KUKA KRL program: SAMPLE.SRC

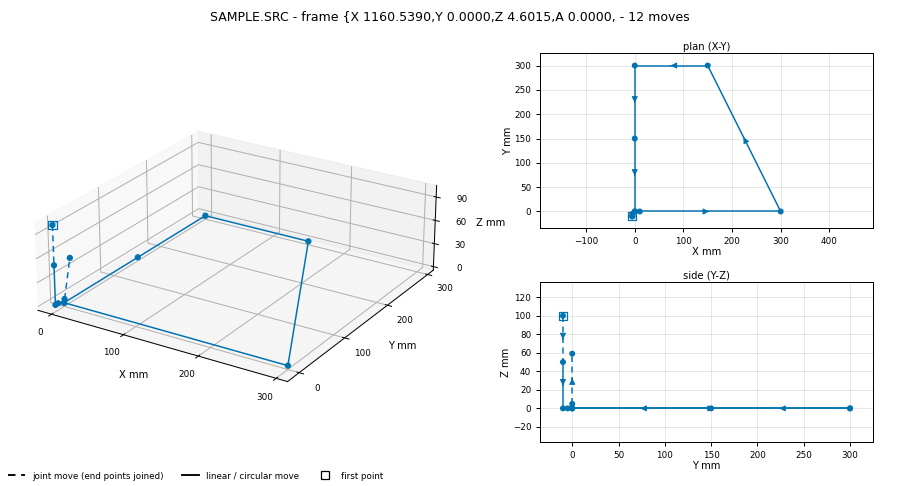
[picture p0: tool path of SAMPLE.SRC in frame {X 1160.5390,Y 0.0000,Z 4.6015,A 0.0000,, 12 of 14 moves have a stored position in this frame; points joined in program order, loops and branches not executed]
&ACCESS RVP
&REL 1
&COMMENT GENERATED BY ROBOTMASTER
&PARAM TEMPLATE = C:\KRC\Roboter\Template\vorgabe
&PARAM EDITMASK = *
DEF BTEST()

EXT BAS (BAS_COMMAND :IN,REAL :IN )
EXT TOOL(INT:IN)
EXT TOOLON()
EXT TOOLOFF()

INT I
BAS (#INITMOV,0 )

;******SETTINGS FOR PTP MOTION***********************
;FOLD
;SET PTP $VEL_AXIS AND $ACC_AXIS
FOR I=1 TO 6
   $VEL_AXIS[I]=50
   $ACC_AXIS[I]=100
ENDFOR
;ENDFOLD (SET PTP $VEL_AXIS AND $ACC_AXIS)

;******SETTINGS FOR LIN AND ARC MOTION***************
;FOLD
;SET LIN AND ARC MOTION VARIABLES
$VEL.CP=0.05
$VEL.ORI1=200
$VEL.ORI2=200
$ACC.ORI1=100
$ACC.ORI2=100
;ENDFOLD (SET LIN AND ARC MOTION VARIABLES)

;******SETTINGS FOR POSITIONING CRITERIA*************
;FOLD
;SET POSITIONING CRITERIA
  $ORI_TYPE = #VAR
;ENDFOLD (SET POSITIONING CRITERIA)

$BASE={X 1160.5390,Y 0.0000,Z 4.6015,A 0.0000,B 0.0000,C 0.0000}
$TOOL={X -352.6447,Y 0.0000,Z 469.2759,A 0.0000,B -60.0005,C 0.0000}

$ADVANCE = 5
PTP  {A1 0.0000,A2 0.0000,A3 0.0000,A4 0.0000,A5 0.0000,A6 0.0000}
TOOL(8)
PTP  {X -5.0000,Y -10.0000,Z 100.0000,A -45.0000,B 0.0000,C 180.0000,S 6,T 54}
PTP  {X -5.0000,Y -10.0000,Z 50.0000,A -45.0000,B 0.0000,C 180.0000,S 6,T 54}
$VEL.CP=0.05  ;50mm/s
LIN  {X -5.0000,Y -10.0000,Z 0.0000,A -45.0000,B 0.0000,C 180.0000}
TOOLON()
LIN  {X -5.0000,Y -5.0000,Z 0.0000,A -45.0000,B 0.0000,C 180.0000}
CIRC {X -3.5355,Y -1.4645,Z 0.0000,A -45.0000,B 0.0000,C 180.0000},{X 0.0000,Y 0.0000,Z 0.0000,A -45.0000,B 0.0000,C 180.0000}
LIN  {X 300.0000,Y 0.0000,Z 0.0000,A -45.0000,B 0.0000,C 180.0000}

(...)

LIN  {X 150.0000,Y 300.0000,Z 0.0000,A -44.5615,B 7.0530,C -172.8929}
LIN  {X 0.0000,Y 300.0000,Z 0.0000,A -45.4385,B 7.0530,C 172.8929}
LIN  {X 0.0000,Y 150.0000,Z 0.0000,A -45.4385,B 7.0530,C 172.8929}
LIN  {X 0.0000,Y 0.0000,Z 0.0000,A -45.4385,B 7.0530,C 172.8929}
TOOLOFF()
PTP  {X 0.8682,Y 0.0000,Z 4.9240,A -45.4385,B 7.0530,C 172.8929,S 6,T 54}
PTP  {X 10.4189,Y 0.0000,Z 59.0885,A -45.4385,B 7.0530,C 172.8929,S 6,T 54}
PTP  {A1 0.0000,A2 0.0000,A3 0.0000,A4 0.0000,A5 0.0000,A6 0.0000}

END
